// TIA Portal project "ASRS" (V17)

(* hardware
DEVICE "S7-1200 station_1"  S7-1200 Station
   slot 0: "Rack_0"  S7-1200 Rack  Rack  V1.0
   slot 1: "PLC_1"  CPU 1212C DC/DC/Rly  6ES7 212-1HE40-0XB0  V4.5
*)

// ===== PLC "PLC_1"  CPU 1212C DC/DC/Rly =====

VAR_GLOBAL   // PLC tag table "Default tag table"
   "Emitter" AT %Q1.0 : Bool;
   "Entry Conveyor" AT %Q1.1 : Bool;
   "Load Conveyor" AT %Q1.2 : Bool;
   "Forks Left" AT %Q1.3 : Bool;
   "Forks Rights" AT %Q1.4 : Bool;
   "Lift" AT %Q1.5 : Bool;
   "Unload Conveyor" AT %Q1.6 : Bool;
   "Exit Conveyor" AT %Q1.7 : Bool;
   "Target Position" AT %QW100 : Int;
   "Start Store" AT %M0.1 : Bool;
   "At Entry" AT %I1.0 : Bool;
   "At Load" AT %I1.1 : Bool;
   "At left" AT %I1.2 : Bool;
   "At middle" AT %I1.3 : Bool;
   "At Right" AT %I1.4 : Bool;
   "At Unload" AT %I1.5 : Bool;
   "At Exit" AT %I1.6 : Bool;
   "Moving X" AT %I1.7 : Bool;
   "Start Initial" AT %M0.0 : Bool;
   "Start Retrieve" AT %M0.2 : Bool;
   "Reset" AT %M0.6 : Bool;
   "Proses Move" AT %M0.7 : Bool;
   "Home" AT %M1.1 : Bool;
   "Store Step1" AT %M2.0 : Bool;
   "Store Step2" AT %M2.1 : Bool;
   "Store Step3" AT %M2.2 : Bool;
   "Store Step4" AT %M2.3 : Bool;
   "Store Step5" AT %M2.4 : Bool;
   "Store Step6" AT %M2.5 : Bool;
   "Store Step7" AT %M2.6 : Bool;
   "Store Step8" AT %M2.7 : Bool;
   "Retrieve Step1" AT %M3.0 : Bool;
   "Retrieve Step2" AT %M3.1 : Bool;
   "Retrieve Step3" AT %M3.2 : Bool;
   "Retrieve Step4" AT %M3.3 : Bool;
   "Retrieve Step5" AT %M3.4 : Bool;
   "Retrieve Step6" AT %M3.5 : Bool;
   "Retrieve Step7" AT %M3.6 : Bool;
   "Retrieve Step8" AT %M3.7 : Bool;
   "Factory Reset" AT %Q2.0 : Bool;
   "Stacker Busy" AT %M0.3 : Bool;
   "id_pallet" AT %IW100 : Int;
END_VAR

DATA_BLOCK "Data_block_1"   // DB10
{ S7_Optimized_Access := 'FALSE' }
VERSION : 0.1
   VAR
      DATA : Array[0..1] of Word;
   END_VAR
BEGIN
END_DATA_BLOCK

// folder: System blocks/Program resources

DATA_BLOCK "IEC_Timer_0_DB"   // DB1
{ S7_Optimized_Access := 'TRUE' }
AUTHOR : Simatic
FAMILY : IEC
NAME : IEC_TMR
VERSION : 1.0
// stored: InstanceOfName IEC_TIMER
"IEC_TIMER"
BEGIN
END_DATA_BLOCK

DATA_BLOCK "IEC_Timer_0_DB_1"   // DB2
{ S7_Optimized_Access := 'TRUE' }
AUTHOR : Simatic
FAMILY : IEC
NAME : IEC_TMR
VERSION : 1.0
// stored: InstanceOfName IEC_TIMER
"IEC_TIMER"
BEGIN
END_DATA_BLOCK

DATA_BLOCK "IEC_Timer_0_DB_2"   // DB3
{ S7_Optimized_Access := 'TRUE' }
AUTHOR : Simatic
FAMILY : IEC
NAME : IEC_TMR
VERSION : 1.0
// stored: InstanceOfName IEC_TIMER
"IEC_TIMER"
BEGIN
END_DATA_BLOCK

DATA_BLOCK "IEC_Timer_0_DB_3"   // DB4
{ S7_Optimized_Access := 'TRUE' }
AUTHOR : Simatic
FAMILY : IEC
NAME : IEC_TMR
VERSION : 1.0
// stored: InstanceOfName IEC_TIMER
"IEC_TIMER"
BEGIN
END_DATA_BLOCK

DATA_BLOCK "IEC_Timer_0_DB_8"   // DB5
{ S7_Optimized_Access := 'TRUE' }
AUTHOR : Simatic
FAMILY : IEC
NAME : IEC_TMR
VERSION : 1.0
// stored: InstanceOfName IEC_TIMER
"IEC_TIMER"
BEGIN
END_DATA_BLOCK

DATA_BLOCK "IEC_Timer_0_DB_4"   // DB6
{ S7_Optimized_Access := 'TRUE' }
AUTHOR : Simatic
FAMILY : IEC
NAME : IEC_TMR
VERSION : 1.0
// stored: InstanceOfName IEC_TIMER
"IEC_TIMER"
BEGIN
END_DATA_BLOCK

DATA_BLOCK "IEC_Timer_0_DB_5"   // DB7
{ S7_Optimized_Access := 'TRUE' }
AUTHOR : Simatic
FAMILY : IEC
NAME : IEC_TMR
VERSION : 1.0
// stored: InstanceOfName IEC_TIMER
"IEC_TIMER"
BEGIN
END_DATA_BLOCK

DATA_BLOCK "IEC_Timer_0_DB_6"   // DB8
{ S7_Optimized_Access := 'TRUE' }
AUTHOR : Simatic
FAMILY : IEC
NAME : IEC_TMR
VERSION : 1.0
// stored: InstanceOfName IEC_TIMER
"IEC_TIMER"
BEGIN
END_DATA_BLOCK

DATA_BLOCK "IEC_Timer_0_DB_7"   // DB9
{ S7_Optimized_Access := 'TRUE' }
AUTHOR : Simatic
FAMILY : IEC
NAME : IEC_TMR
VERSION : 1.0
// stored: InstanceOfName IEC_TIMER
"IEC_TIMER"
BEGIN
END_DATA_BLOCK

DATA_BLOCK "IEC_Timer_0_DB_9"   // DB11
{ S7_Optimized_Access := 'TRUE' }
AUTHOR : Simatic
FAMILY : IEC
NAME : IEC_TMR
VERSION : 1.0
// stored: InstanceOfName IEC_TIMER
"IEC_TIMER"
BEGIN
END_DATA_BLOCK

DATA_BLOCK "IEC_Timer_0_DB_10"   // DB12
{ S7_Optimized_Access := 'TRUE' }
AUTHOR : Simatic
FAMILY : IEC
NAME : IEC_TMR
VERSION : 1.0
// stored: InstanceOfName IEC_TIMER
"IEC_TIMER"
BEGIN
END_DATA_BLOCK

DATA_BLOCK "IEC_Timer_0_DB_11"   // DB13
{ S7_Optimized_Access := 'TRUE' }
AUTHOR : Simatic
FAMILY : IEC
NAME : IEC_TMR
VERSION : 1.0
// stored: InstanceOfName IEC_TIMER
"IEC_TIMER"
BEGIN
END_DATA_BLOCK

DATA_BLOCK "IEC_Timer_0_DB_12"   // DB14
{ S7_Optimized_Access := 'TRUE' }
AUTHOR : Simatic
FAMILY : IEC
NAME : IEC_TMR
VERSION : 1.0
// stored: InstanceOfName IEC_TIMER
"IEC_TIMER"
BEGIN
END_DATA_BLOCK

DATA_BLOCK "IEC_Timer_0_DB_13"   // DB15
{ S7_Optimized_Access := 'TRUE' }
AUTHOR : Simatic
FAMILY : IEC
NAME : IEC_TMR
VERSION : 1.0
// stored: InstanceOfName IEC_TIMER
"IEC_TIMER"
BEGIN
END_DATA_BLOCK

DATA_BLOCK "IEC_Timer_0_DB_14"   // DB16
{ S7_Optimized_Access := 'TRUE' }
AUTHOR : Simatic
FAMILY : IEC
NAME : IEC_TMR
VERSION : 1.0
// stored: InstanceOfName IEC_TIMER
"IEC_TIMER"
BEGIN
END_DATA_BLOCK

DATA_BLOCK "IEC_Timer_0_DB_15"   // DB17
{ S7_Optimized_Access := 'TRUE' }
AUTHOR : Simatic
FAMILY : IEC
NAME : IEC_TMR
VERSION : 1.0
// stored: InstanceOfName IEC_TIMER
"IEC_TIMER"
BEGIN
END_DATA_BLOCK

DATA_BLOCK "IEC_Timer_0_DB_16"   // DB18
{ S7_Optimized_Access := 'TRUE' }
AUTHOR : Simatic
FAMILY : IEC
NAME : IEC_TMR
VERSION : 1.0
// stored: InstanceOfName IEC_TIMER
"IEC_TIMER"
BEGIN
END_DATA_BLOCK

// folder: (top level)

ORGANIZATION_BLOCK "Warehouse"   // OB1, LAD, ProgramCycle
TITLE = "Main Program Sweep (Cycle)"
{ S7_Optimized_Access := 'TRUE' }
VERSION : 0.1
// For ASRS simulation in Factory IO
   VAR_INPUT
      Initial_Call : Bool;   // Initial call of this OB
      Remanence : Bool;   // =True, if remanent data are available
   END_VAR
   VAR_TEMP   // added for the SCL form of the ladder/FBD networks
      _w1 : Bool;
   END_VAR
BEGIN

REGION Network 1: Supply Pallet
   // Initial pallet, start to emitter
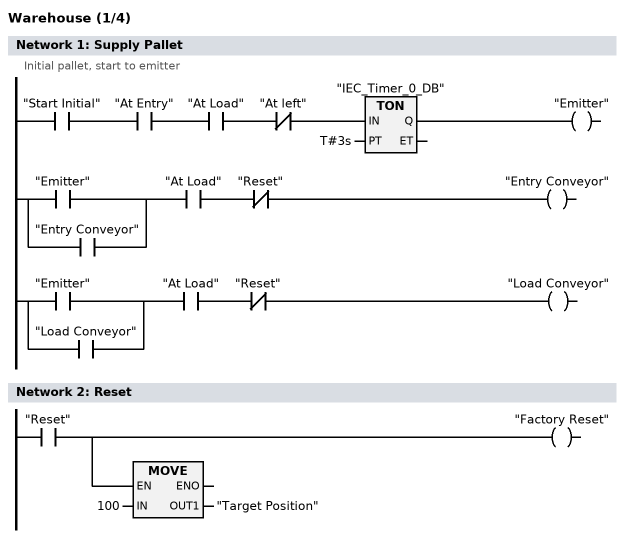
   "IEC_Timer_0_DB".TON(IN := "Start Initial" AND "At Entry" AND "At Load" AND NOT "At left", PT := T#3s);
   "Emitter" := "IEC_Timer_0_DB".Q;
   "Entry Conveyor" := ("Emitter" OR "Entry Conveyor") AND "At Load" AND NOT "Reset";
   "Load Conveyor" := ("Emitter" OR "Load Conveyor") AND "At Load" AND NOT "Reset";
END_REGION

REGION Network 2: Reset
   RUNG wire#powerrail
      Contact( "Reset" )
      wire#w1
      Coil( "Factory Reset" )
   END_RUNG
   RUNG wire#w1
      Move(in := 100, out1 => "Target Position")
   END_RUNG
   // the same network as SCL:
   "Factory Reset" := "Reset";
   IF "Reset" THEN "Target Position" := 100; END_IF;
END_REGION

REGION Network 3: Start Store Pallet to Rack
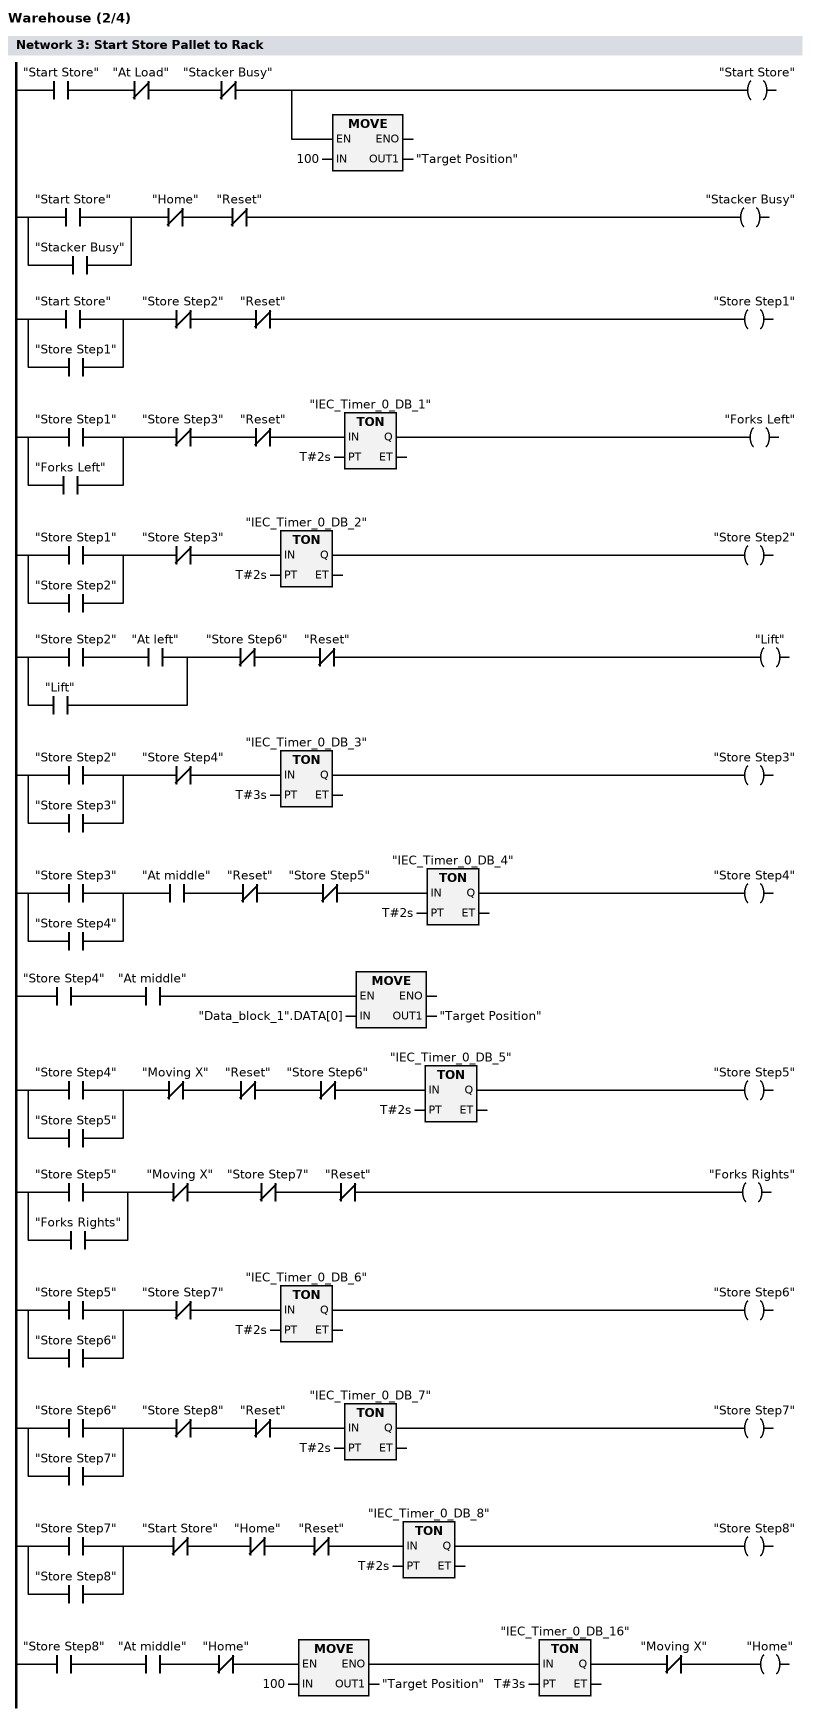
   "Start Store" := "Start Store" AND NOT "At Load" AND NOT "Stacker Busy";
   IF "Start Store" THEN "Target Position" := 100; END_IF;
   "Stacker Busy" := ("Start Store" OR "Stacker Busy") AND NOT "Home" AND NOT "Reset";
   "Store Step1" := ("Start Store" OR "Store Step1") AND NOT "Store Step2" AND NOT "Reset";
   "IEC_Timer_0_DB_1".TON(IN := ("Store Step1" OR "Forks Left") AND NOT "Store Step3" AND NOT "Reset",
                          PT := T#2s);
   "Forks Left" := "IEC_Timer_0_DB_1".Q;
   "IEC_Timer_0_DB_2".TON(IN := ("Store Step1" OR "Store Step2") AND NOT "Store Step3", PT := T#2s);
   "Store Step2" := "IEC_Timer_0_DB_2".Q;
   "Lift" := (("Store Step2" AND "At left") OR "Lift") AND NOT "Store Step6" AND NOT "Reset";
   "IEC_Timer_0_DB_3".TON(IN := ("Store Step2" OR "Store Step3") AND NOT "Store Step4", PT := T#3s);
   "Store Step3" := "IEC_Timer_0_DB_3".Q;
   "IEC_Timer_0_DB_4".TON(IN := ("Store Step3" OR "Store Step4") AND "At middle" AND NOT "Reset" AND NOT "Store Step5",
                          PT := T#2s);
   "Store Step4" := "IEC_Timer_0_DB_4".Q;
   IF "Store Step4" AND "At middle" THEN "Target Position" := "Data_block_1".DATA[0]; END_IF;
   "IEC_Timer_0_DB_5".TON(IN := ("Store Step4" OR "Store Step5") AND NOT "Moving X" AND NOT "Reset" AND NOT "Store Step6",
                          PT := T#2s);
   "Store Step5" := "IEC_Timer_0_DB_5".Q;
   "Forks Rights" := ("Store Step5" OR "Forks Rights") AND NOT "Moving X" AND NOT "Store Step7" AND NOT "Reset";
   "IEC_Timer_0_DB_6".TON(IN := ("Store Step5" OR "Store Step6") AND NOT "Store Step7", PT := T#2s);
   "Store Step6" := "IEC_Timer_0_DB_6".Q;
   "IEC_Timer_0_DB_7".TON(IN := ("Store Step6" OR "Store Step7") AND NOT "Store Step8" AND NOT "Reset",
                          PT := T#2s);
   "Store Step7" := "IEC_Timer_0_DB_7".Q;
   "IEC_Timer_0_DB_8".TON(IN := ("Store Step7" OR "Store Step8") AND NOT "Start Store" AND NOT "Home" AND NOT "Reset",
                          PT := T#2s);
   "Store Step8" := "IEC_Timer_0_DB_8".Q;
   #_w1 := "Store Step8" AND "At middle" AND NOT "Home";
   IF #_w1 THEN "Target Position" := 100; END_IF;
   "IEC_Timer_0_DB_16".TON(IN := #_w1, PT := T#3s);
   "Home" := "IEC_Timer_0_DB_16".Q AND NOT "Moving X";
END_REGION

REGION Network 4: Start to Retrieve
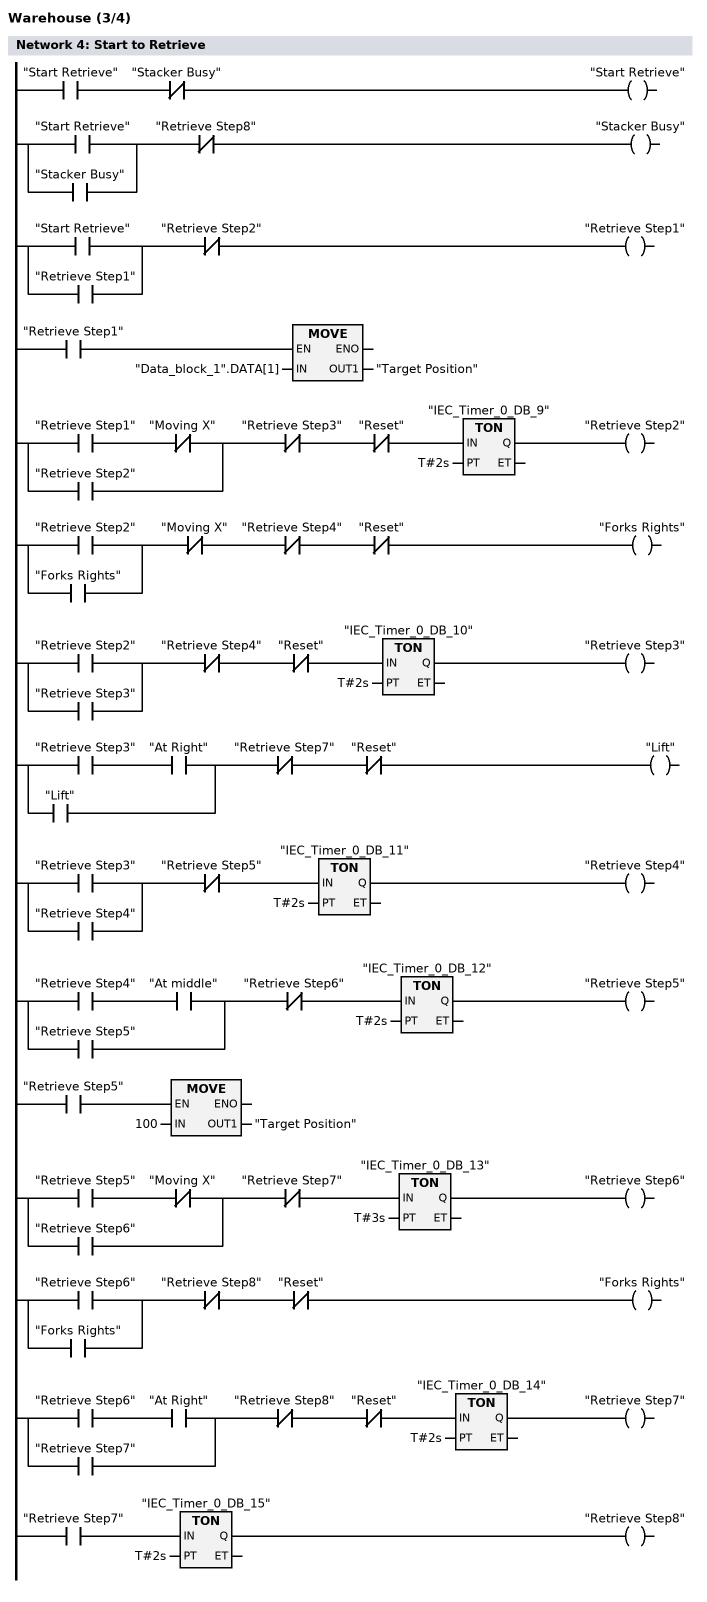
   "Start Retrieve" := "Start Retrieve" AND NOT "Stacker Busy";
   "Stacker Busy" := ("Start Retrieve" OR "Stacker Busy") AND NOT "Retrieve Step8";
   "Retrieve Step1" := ("Start Retrieve" OR "Retrieve Step1") AND NOT "Retrieve Step2";
   IF "Retrieve Step1" THEN "Target Position" := "Data_block_1".DATA[1]; END_IF;
   "IEC_Timer_0_DB_9".TON(IN := (("Retrieve Step1" AND NOT "Moving X") OR "Retrieve Step2") AND NOT "Retrieve Step3" AND NOT "Reset",
                          PT := T#2s);
   "Retrieve Step2" := "IEC_Timer_0_DB_9".Q;
   "Forks Rights" := ("Retrieve Step2" OR "Forks Rights") AND NOT "Moving X" AND NOT "Retrieve Step4" AND NOT "Reset";
   "IEC_Timer_0_DB_10".TON(IN := ("Retrieve Step2" OR "Retrieve Step3") AND NOT "Retrieve Step4" AND NOT "Reset",
                           PT := T#2s);
   "Retrieve Step3" := "IEC_Timer_0_DB_10".Q;
   "Lift" := (("Retrieve Step3" AND "At Right") OR "Lift") AND NOT "Retrieve Step7" AND NOT "Reset";
   "IEC_Timer_0_DB_11".TON(IN := ("Retrieve Step3" OR "Retrieve Step4") AND NOT "Retrieve Step5", PT := T#2s);
   "Retrieve Step4" := "IEC_Timer_0_DB_11".Q;
   "IEC_Timer_0_DB_12".TON(IN := (("Retrieve Step4" AND "At middle") OR "Retrieve Step5") AND NOT "Retrieve Step6",
                           PT := T#2s);
   "Retrieve Step5" := "IEC_Timer_0_DB_12".Q;
   IF "Retrieve Step5" THEN "Target Position" := 100; END_IF;
   "IEC_Timer_0_DB_13".TON(IN := (("Retrieve Step5" AND NOT "Moving X") OR "Retrieve Step6") AND NOT "Retrieve Step7",
                           PT := T#3s);
   "Retrieve Step6" := "IEC_Timer_0_DB_13".Q;
   "Forks Rights" := ("Retrieve Step6" OR "Forks Rights") AND NOT "Retrieve Step8" AND NOT "Reset";
   "IEC_Timer_0_DB_14".TON(IN := (("Retrieve Step6" AND "At Right") OR "Retrieve Step7") AND NOT "Retrieve Step8" AND NOT "Reset",
                           PT := T#2s);
   "Retrieve Step7" := "IEC_Timer_0_DB_14".Q;
   "IEC_Timer_0_DB_15".TON(IN := "Retrieve Step7", PT := T#2s);
   "Retrieve Step8" := "IEC_Timer_0_DB_15".Q;
END_REGION

REGION Network 5: Unload Conveyor
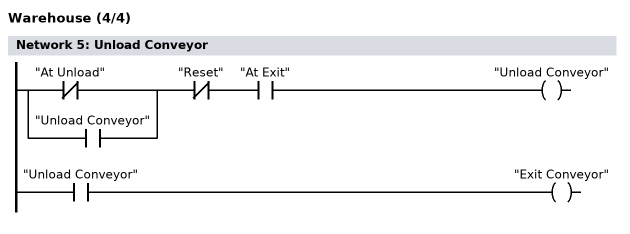
   RUNG wire#powerrail
      I_Contact( "At Unload" )
      wire#w1
      I_Contact( "Reset" )
      Contact( "At Exit" )
      Coil( "Unload Conveyor" )
   END_RUNG
   RUNG wire#powerrail
      Contact( "Unload Conveyor" )
   END_RUNG wire#w1
   RUNG wire#powerrail
      Contact( "Unload Conveyor" )
      Coil( "Exit Conveyor" )
   END_RUNG
   // the same network as SCL:
   "Unload Conveyor" := (NOT "At Unload" OR "Unload Conveyor") AND NOT "Reset" AND "At Exit";
   "Exit Conveyor" := "Unload Conveyor";
END_REGION
END_ORGANIZATION_BLOCK